Fanuc KAREL source: test_layout.kl

PROGRAM test_layout
%NOLOCKGROUP

%include systemlib.types.klt
%include systemlib.datatypes.klt
%include pathlib.klt
%include pose.const.klt

CONST
  FILE_NAME = 'FR:test3599.csv'
VAR
  eof : BOOLEAN
  buffernum FROM tstlay: INTEGER
  passes : PATH nodedata = t_INTEGER
  layers : INTEGER

%include display.klh

-- layout object
%class tstlay('pathlayout.klc','pathlayout.klh','defaultpathlayout.klt')


ROUTINE clear_list
  VAR
    i : INTEGER
    status : INTEGER
  BEGIN
    i = PATH_LEN(passes)
    WHILE PATH_LEN(passes) > 0 DO
		  DELETE_NODE(passes,i,status)
      i = i - 1
	  ENDWHILE
  END clear_list

ROUTINE print_list
  VAR
    i : INTEGER
  BEGIN
    FOR i=1 TO PATH_LEN(passes) DO
      WRITE TPDISPLAY('L',i,': ', passes[i].v, ' passes', CR)
    ENDFOR
  END print_list

BEGIN
  --clear display
  display__clear
  --show display
  display__show

  clear_list

  --construct
  tstlay__new(FILE_NAME, PTH_CARTESAN, Z_AXES)

  -- ** predetermine number of layers and passes in each layer **

  --get numbers of layers
  tstlay__openfile

  --count the number of passes per layer
  tstlay__countInstances(passes)

  --get number of layers
  layers = PATH_LEN(passes)

  --print
  WRITE TPDISPLAY('total Layers: ', layers, CR)
  print_list


  tstlay__closefile

  -- ** Load layers into a path buffer **

  tstlay__openfile

  --load per layer
  REPEAT
    eof = tstlay__loadBuffer
    WRITE TPDISPLAY('L', buffernum, ': eof', eof, ',', tstlay__bufferLength, ' nodes', CR)
  UNTIL(eof)

  tstlay__closefile

  --delete
  --tstlay__delete

END test_layout
